PROGRAM MAIN_LINE2
VAR
	traError			: BOOL;
	traInitDone			: BOOL;
	bModeOff			: BOOL;
	bModeManual			: BOOL := TRUE;
	bModeAuto			: BOOL;
	Err_T				: R_TRIG;
	Wrn_T				: R_TRIG;
	fbtimer				: TON;
	fbTimerSirens		: TON;
	Run_T				: R_TRIG;
	Stop_T				: R_TRIG;
	k,k1				: INT;
	nState				: INT;
	nState1				: INT;
	nStateEmr			: INT;
	bFaultFlag			: BOOL;
	nstateStop			: INT;
	fbTimerStop			: TON;
	timerStop			: ton;
	timerReset			: TON;
	thne				: INT;
	nState2				: INT;
	Reset_T				: R_TRIG;
	fbEventlogger		: FB_Eventlogger;
	bWriteAlarm			: BOOL;
END_VAR

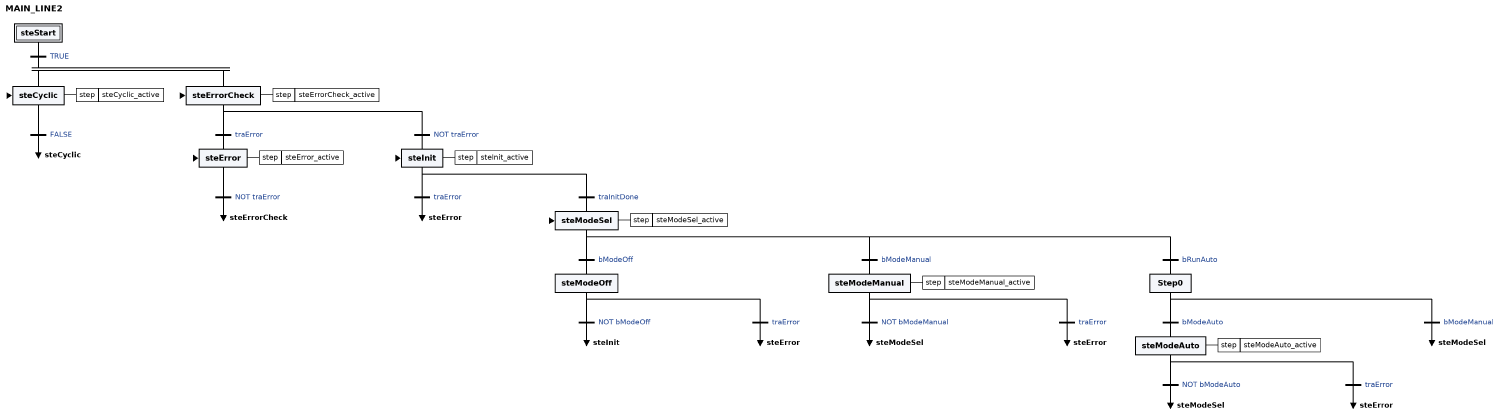
INITIAL_STEP steStart:
END_STEP
TRANSITION FROM steStart TO (steCyclic, steErrorCheck)
    := TRUE;
END_TRANSITION
STEP steCyclic:
    steCyclic_active(N);  // step action
END_STEP
TRANSITION FROM steCyclic TO steCyclic
    := FALSE;
END_TRANSITION
STEP steErrorCheck:
    steErrorCheck_active(N);  // step action
END_STEP
TRANSITION FROM steErrorCheck TO steError
    := traError;
END_TRANSITION
STEP steError:
    steError_active(N);  // step action
END_STEP
TRANSITION FROM steError TO steErrorCheck
    := NOT traError;
END_TRANSITION
TRANSITION FROM steErrorCheck TO steInit
    := NOT traError;
END_TRANSITION
STEP steInit:
    steInit_active(N);  // step action
END_STEP
TRANSITION FROM steInit TO steError
    := traError;
END_TRANSITION
TRANSITION FROM steInit TO steModeSel
    := traInitDone;
END_TRANSITION
STEP steModeSel:
    steModeSel_active(N);  // step action
END_STEP
TRANSITION FROM steModeSel TO steModeOff
    := bModeOff;
END_TRANSITION
STEP steModeOff:
END_STEP
TRANSITION FROM steModeOff TO steInit
    := NOT bModeOff;
END_TRANSITION
TRANSITION FROM steModeOff TO steError
    := traError;
END_TRANSITION
TRANSITION FROM steModeSel TO steModeManual
    := bModeManual;
END_TRANSITION
STEP steModeManual:
    steModeManual_active(N);  // step action
END_STEP
TRANSITION FROM steModeManual TO steModeSel
    := NOT bModeManual;
END_TRANSITION
TRANSITION FROM steModeManual TO steError
    := traError;
END_TRANSITION
TRANSITION FROM steModeSel TO Step0
    := bRunAuto;
END_TRANSITION
STEP Step0:
END_STEP
TRANSITION FROM Step0 TO steModeAuto
    := bModeAuto;
END_TRANSITION
TRANSITION FROM Step0 TO steModeSel
    := bModeManual;
END_TRANSITION
STEP steModeAuto:
    steModeAuto_active(N);  // step action
END_STEP
TRANSITION FROM steModeAuto TO steModeSel
    := NOT bModeAuto;
END_TRANSITION
TRANSITION FROM steModeAuto TO steError
    := traError;
END_TRANSITION

ACTION ListError:
Err_T(CLK := bError2);
Wrn_T(CLK := bWarning2);
GetLocalSystemTime(bEnable := 1,);
IF a2 > 100 THEN
	a2 := 100;
END_IF
		
CASE nState OF 
	0:
		IF Err_T.Q THEN
			nState := 1;
		ELSIF Wrn_T.Q THEN
			bWrn2 := true;
			nState := 10;
		END_IF
	1:
		CASE nErrorID OF	
			23:
				stErrorTxt2 := "E1_2.Lỗi hết hũ trạm 2 [kiểm tra U1I2-4]";
				stErrorTxt3 := 'E1_2.The jar is empty line 2 [check U1I2-4]';
				fbEventlogger(eventClass := TC_EVENTS.Entobel.Event23.uuidEventClass, nEventID := DINT_TO_UDINT(nErrorID));
			24:
				stErrorTxt2 := "E2_2.Lỗi hũ bị kẹt trạm 2 [kiểm tra U1I2-8]";
				stErrorTxt3 := 'E2_2.The jar  is trapped line 2 [check U1I2-8]';
				fbEventlogger(eventClass := TC_EVENTS.Entobel.Event24.uuidEventClass, nEventID := DINT_TO_UDINT(nErrorID));
			25:
				stErrorTxt2 := "E3_2.Lỗi ben chặn hũ trên rút về trạm 2 [kiểm tra U1I2-5]" ;
				stErrorTxt3 := 'E3_2.The upper cylinder retract  is faulty line 2 [check U1I2-5]';
				fbEventlogger(eventClass := TC_EVENTS.Entobel.Event25.uuidEventClass, nEventID := DINT_TO_UDINT(nErrorID));
			26:
				stErrorTxt2 := "E4_2.Lỗi ben chặn hũ dưới rút về trạm 2 [kiểm tra U1I2-6]";
				stErrorTxt3 := 'E4_2.The lower cylinder retract  is faulty line 2 [check U1I2-6]';
				fbEventlogger(eventClass := TC_EVENTS.Entobel.Event26.uuidEventClass, nEventID := DINT_TO_UDINT(nErrorID));
			27:
				stErrorTxt2 := "E5_2.Lỗi ben chặn hũ dưới đẩy ra trạm 2 [kiểm tra U1I2-7]";
				stErrorTxt3 := 'E5_2.The lower cylinder extend  is faulty line 2 [check U1I2-7]';
				fbEventlogger(eventClass := TC_EVENTS.Entobel.Event27.uuidEventClass, nEventID := DINT_TO_UDINT(nErrorID));
			28:
				stErrorTxt2 := "E6_2.Lỗi biến tần đảo thức ăn trạm 2 [kiểm tra biến tần 1]";
				stErrorTxt3 := 'E6_2.The inverter of agitator motor fault line 2 [check inverter 1]';
				fbEventlogger(eventClass := TC_EVENTS.Entobel.Event28.uuidEventClass, nEventID := DINT_TO_UDINT(nErrorID));
			29:
				stErrorTxt2 := "E7_2.Lỗi driver chia thức ăn trạm 2 [kiểm tra driver 1]";
				stErrorTxt3 := 'E7_2.The driver of dispenser motor fault line 2 [check driver 1]';
				fbEventlogger(eventClass := TC_EVENTS.Entobel.Event29.uuidEventClass, nEventID := DINT_TO_UDINT(nErrorID));
			30:
				stErrorTxt2 := "E8_2.Lỗi ben chặn sâu rút về trạm 2 [kiểm tra U1I3-1]";
				stErrorTxt3 := 'E8_2.The cylinder blocking worm retract is faulty line 2 [check U1I3-1]';
				fbEventlogger(eventClass := TC_EVENTS.Entobel.Event30.uuidEventClass, nEventID := DINT_TO_UDINT(nErrorID));
			31:
				stErrorTxt2 := "E9_2.Lỗi biến tần phểu rung sâu trạm 2 [kiểm tra biến tần 2]";
				stErrorTxt3 := 'E9_2.The inverter of vibrating funnel fault line 2 [check inverter 2]';
				fbEventlogger(eventClass := TC_EVENTS.Entobel.Event31.uuidEventClass, nEventID := DINT_TO_UDINT(nErrorID));
			32:
				stErrorTxt2 := "E10_2.Lỗi hết nắp trạm 2 [kiểm tra U1I3-2]";
				stErrorTxt3 := 'E10_2.The lid is empty line 2 [check U1I3-2]';
				fbEventlogger(eventClass := TC_EVENTS.Entobel.Event32.uuidEventClass, nEventID := DINT_TO_UDINT(nErrorID));
			33:
				stErrorTxt2 := "E11_2.Lỗi ben chặn nắp rút về trạm 2 [kiểm tra U1I3-3]";
				stErrorTxt3 := 'E11_2.The cylinder blocking the lid retract is faulty line 2 [check U1I3-3]';
				fbEventlogger(eventClass := TC_EVENTS.Entobel.Event33.uuidEventClass, nEventID := DINT_TO_UDINT(nErrorID));
			34:
				stErrorTxt2 := "E12_2.Lỗi ben chặn nắp đẩy ra trạm 2 [kiểm tra U1I3-4]";
				stErrorTxt3 := 'E12_2.The cylinder blocking the lid extend is faulty line 2 [check U1I3-4]';
				fbEventlogger(eventClass := TC_EVENTS.Entobel.Event34.uuidEventClass, nEventID := DINT_TO_UDINT(nErrorID));
			35:
				stErrorTxt2 := "E13_2.Lỗi ben hút/thả nắp rút ra trạm 2 [kiểm tra U1I3-5]";
				stErrorTxt3 := 'E13_2.The cylinder sucking the lid retract is faulty line 2 [check U1I3-5]';
				fbEventlogger(eventClass := TC_EVENTS.Entobel.Event35.uuidEventClass, nEventID := DINT_TO_UDINT(nErrorID));
			36:
				stErrorTxt2 := "E14_2.Lỗi ben hút/thả nắp đẩy ra trạm 2 [kiểm tra U1I3-6]";
				stErrorTxt3 := 'E14_2.The cylinder sucking the lid extend is faulty line 2 [check U1I3-6]';
				fbEventlogger(eventClass := TC_EVENTS.Entobel.Event36.uuidEventClass, nEventID := DINT_TO_UDINT(nErrorID));
			37:
				stErrorTxt2 := "E15_2.Lỗi ben dập nắp rút về trạm 2 [kiểm tra U1I3-8]";
				stErrorTxt3 := 'E15_2.The cylinder pressing the lid retract is faulty line 2 [check U1I3-8]';
				fbEventlogger(eventClass := TC_EVENTS.Entobel.Event37.uuidEventClass, nEventID := DINT_TO_UDINT(nErrorID));
			38:
				stErrorTxt2 := "E16_2.Lỗi ben dập nắp đẩy ra trạm 2 [kiểm tra U1I4-1]";
				stErrorTxt3 := 'E16_2.The cylinder pressing the lid extend is faulty line 2 [check U1I4-1]';
				fbEventlogger(eventClass := TC_EVENTS.Entobel.Event38.uuidEventClass, nEventID := DINT_TO_UDINT(nErrorID));
			39:
				stErrorTxt2 := "E17_2.Lỗi ben lượt ra/vào Rút về trạm 2 [kiểm tra U1I4-2]";
				stErrorTxt3 := 'E17_2.The comb cylinder retract is faulty line 2 [check U1I4-2]';
				fbEventlogger(eventClass := TC_EVENTS.Entobel.Event39.uuidEventClass, nEventID := DINT_TO_UDINT(nErrorID));
			40:
				stErrorTxt2 := "E18_2.Lỗi ben lượt ra/vào đẩy ra trạm 2 [kiểm tra U1I4-3]";
				stErrorTxt3 := 'E18_2.The comb cylinder extend is faulty line 2 [check U1I4-3]';
				fbEventlogger(eventClass := TC_EVENTS.Entobel.Event40.uuidEventClass, nEventID := DINT_TO_UDINT(nErrorID));
			41:
				stErrorTxt2 := "E19_2.Lỗi ben kẹp hũ rút về trạm 2 [kiểm tra U1I4-6]";
				stErrorTxt3 := 'E19_2.The clap cylinder retract is faulty line 2 [check U1I4-6]';
				fbEventlogger(eventClass := TC_EVENTS.Entobel.Event41.uuidEventClass, nEventID := DINT_TO_UDINT(nErrorID));
			42:
				stErrorTxt2 := "E20_2.Lỗi ben kẹp hũ đẩy ra trạm 2 [kiểm tra U1I4-7]";	
				stErrorTxt3 := 'E20_2.The clap cylinder extend is faulty 2 [check U1I4-4]';
				fbEventlogger(eventClass := TC_EVENTS.Entobel.Event42.uuidEventClass, nEventID := DINT_TO_UDINT(nErrorID));
			43:
				stErrorTxt2 := "E21_2.Lỗi ben di chuyển lượt rút về trạm 2 [kiểm tra U1I4-4]";	
				stErrorTxt3 := 'E21_2.The cylinder moving comb retract is faulty line 2 [check U1I4-4]';
				fbEventlogger(eventClass := TC_EVENTS.Entobel.Event43.uuidEventClass, nEventID := DINT_TO_UDINT(nErrorID));
			44:
				stErrorTxt2 := "E22_2.Lỗi ben di chuyển lượt đẩy ra trạm 2 [kiểm tra U1I4-5]";	
				stErrorTxt3 := 'E22_2.The cylinder moving comb extend is faulty line 2 [check U1I4-5]';
				fbEventlogger(eventClass := TC_EVENTS.Entobel.Event44.uuidEventClass, nEventID := DINT_TO_UDINT(nErrorID));
			46:
				stErrorTxt2 := "E23_2.Lỗi mất hũ khi đang cân thức ăn trạm 2 [kiểm tra U1I4-8]";
				stErrorTxt3 := 'E23_2.The jar is missed when weighting food line 2 [check U1I4-8]';
				fbEventlogger(eventClass := TC_EVENTS.Entobel.Event46.uuidEventClass, nEventID := DINT_TO_UDINT(nErrorID));
			48:
				stErrorTxt2 := "E24_2.Lỗi mất hũ khi đang cân sâu trạm 2 [kiểm tra U1I5-1]";
				stErrorTxt3 := 'E24_2.The jar is missed when weighting larvae line 2 [check U1I5-1]';
				fbEventlogger(eventClass := TC_EVENTS.Entobel.Event48.uuidEventClass, nEventID := DINT_TO_UDINT(nErrorID));
			50:
				stErrorTxt2 := "E25_2.Lỗi hút không được nắp trạm 2 [kiểm tra U1I3-7]";
				stErrorTxt3 := 'E25_2.Failed to suction the lid  line 2 [check U1I3-7]';
				fbEventlogger(eventClass := TC_EVENTS.Entobel.Event50.uuidEventClass, nEventID := DINT_TO_UDINT(nErrorID));
			52:
				stErrorTxt2 := "E26_2.Lỗi nắp đã được hút 2 [kiểm tra U1I3-7]";	
				stErrorTxt3 := 'E26_2.The lid is still on the valve line 2 [check U1I3-7]';
				fbEventlogger(eventClass := TC_EVENTS.Entobel.Event52.uuidEventClass, nEventID := DINT_TO_UDINT(nErrorID));
			53:
				stErrorTxt2 := "E27_2.Lỗi an toàn cửa 1 [kiểm tra U1I7-8]";	
				stErrorTxt3 := 'E27_2.The safety door 1 is error [check U1I7-8]';
			54:
				stErrorTxt2 := "E28_2.Lỗi an toàn cửa 2 [kiểm tra U1I7-9]";
				stErrorTxt3 := 'E28_2.The safety door 2 is error [check U1I7-9]';
			55:
				stErrorTxt2 := "E29_2.Lỗi an toàn cửa 3 [kiểm tra U1I7-10]";
				stErrorTxt3 := 'E29_2.The safety door 3 is error [check U1I7-10]';
			58: 
				stErrorTxt2 := "E30_2.Lỗi quá cân thức ăn trạm 2 [kiểm tra cân thức ăn]";
				stErrorTxt3 := 'E30_2.Overload weightfood line 2 [check weightfood]';
				fbEventlogger(eventClass := TC_EVENTS.Entobel.Event58.uuidEventClass, nEventID := DINT_TO_UDINT(nErrorID));
			59: 
				stErrorTxt2 := "E31_2.Lỗi quá cân sâu trạm 2 [kiểm tra cân sâu]";
				stErrorTxt3 := 'E31_2.Overload weightlarvae line 2 [check weightlarvae]';
				fbEventlogger(eventClass := TC_EVENTS.Entobel.Event59.uuidEventClass, nEventID := DINT_TO_UDINT(nErrorID));
			61:
				stErrorTxt2 := "E32_2.Lỗi ben hút/thả hũ đẩy ra trạm 2 [kiểm tra U1I7-12]";
				stErrorTxt3 := 'E32_2.The cylinder sucking the jar is faulty line 2 [check U1I7-12]';
				fbEventlogger(eventClass := TC_EVENTS.Entobel.Event61.uuidEventClass, nEventID := DINT_TO_UDINT(nErrorID));
			62:
				stErrorTxt2 := "E33_2.Lỗi Modbus thiết bị 1";
				stErrorTxt3 := 'E33_2.Error Modbus device 1';
				fbEventlogger(eventClass := TC_EVENTS.Entobel.Event62.uuidEventClass, nEventID := DINT_TO_UDINT(nErrorID));
			63:
				stErrorTxt2 := "E34_2.Lỗi Modbus thiết bị 2";
				stErrorTxt3 := 'E34_2.Error Modbus device 2';
				fbEventlogger(eventClass := TC_EVENTS.Entobel.Event63.uuidEventClass, nEventID := DINT_TO_UDINT(nErrorID));
			64:
				stErrorTxt2 := "E35_2.Lỗi Modbus thiết bị 3";
				stErrorTxt3 := 'E35_2.Error Modbus device 3';
			67:
				stErrorTxt2 := "E36_2.Lỗi Modbus thiết bị 6";
				stErrorTxt3 := 'E36_2.Error Modbus device 6';
				fbEventlogger(eventClass := TC_EVENTS.Entobel.Event67.uuidEventClass, nEventID := DINT_TO_UDINT(nErrorID));
			71:
				stErrorTxt2 := "E37_2.Lỗi đầu cân thức ăn Laumas";
				stErrorTxt3 := 'E37_2.Error Laumas 1';
				fbEventlogger(eventClass := TC_EVENTS.Entobel.Event71.uuidEventClass, nEventID := DINT_TO_UDINT(nErrorID));
			72:
				stErrorTxt2 := "E38_2.Lỗi đầu cân sâu Laumas";
				stErrorTxt3 := 'E38_2.Error Laumas 2';
				fbEventlogger(eventClass := TC_EVENTS.Entobel.Event72.uuidEventClass, nEventID := DINT_TO_UDINT(nErrorID));
			74:
				stErrorTxt2 := "E39_2.Lỗi ben chặn sâu đẩy ra trạm 2 [kiểm tra U1I3-1]";
				stErrorTxt3 := 'E39_2.The cylinder blocking worm extend  is faulty line 2';
				fbEventlogger(eventClass := TC_EVENTS.Entobel.Event74.uuidEventClass, nEventID := DINT_TO_UDINT(nErrorID));
			75:
				stErrorTxt2 := "E40_2.Lỗi thiếu khí đầu vào [kiểm tra U1I7-13]";
				stErrorTxt3 := 'E40_2.Error of lack of input air [check U1I7-13]';	
			78:
				stErrorTxt2 := "E41_2.Lỗi hết thức ăn trạm 2";
				stErrorTxt3 := 'E41_2.Error running out of food line 2';
				fbEventlogger(eventClass := TC_EVENTS.Entobel.Event77.uuidEventClass, nEventID := DINT_TO_UDINT(nErrorID));	
			79:
				stErrorTxt2 := "E42_2.Lỗi hết sâu trạm 2";
				stErrorTxt3 := 'E42_2.Error running out of larvae line 2';
				fbEventlogger(eventClass := TC_EVENTS.Entobel.Event79.uuidEventClass, nEventID := DINT_TO_UDINT(nErrorID));	
			98:
				stErrorTxt2 := "E98_2.Dừng khẩn [kiểm tra Emergency]"; 
				stErrorTxt3 := 'E98_2.Emergency Stop [check Emergency]';
			99: 
				stErrorTxt2 := "E99_2.Lỗi biến tần băng tải đầu ra [kiểm tra biến tần 3]";
				stErrorTxt3 := 'E99_2.The inverter of conveyor ouy [check inverter 3]';
		END_CASE
		IF a2 <> 1 THEN
			FOR	k := a2 TO 2 BY -1 DO
				nErrorIDList2[k].nErrorID 	 := nErrorIDList2[k-1].nErrorID;
				nErrorIDList2[k].ErrorTime   := nErrorIDList2[k-1].ErrorTime;
				nErrorIDList2[k].ErrorStatus := nErrorIDList2[k-1].ErrorStatus;	
			END_FOR		
		END_IF 
		nErrorIDList2[1].nErrorID := nErrorID;
		nErrorIDList2[1].ErrorTime := SYSTEMTIME_TO_DT(GetLocalSystemTime.systemTime);
		nErrorIDList2[1].ErrorStatus := 1;
		nStatus2	:= 'ERROR';
		a2 := a2 + 1;
		bWarning := FALSE;
		nState := 2;
	2:
		bWriteAlarm	:= TRUE;
		IF nErrorID = 53 THEN
			bTo_alarm_side2 := FALSE;
		ELSIF nErrorID = 54 THEN
			bTo_alarm_side2 := FALSE;
		ELSIF nErrorID = 55 THEN
			bTo_alarm_side2 := FALSE;
		ELSIF nErrorID = 64 THEN
			bTo_alarm_side2 := FALSE;
		ELSIF nErrorID = 75 THEN
			bTo_alarm_side2 := FALSE;
		ELSIF nErrorID = 98 THEN
			bTo_alarm_side2 := FALSE;
		ELSIF nErrorID = 99 THEN
			bTo_alarm_side2 := FALSE;
		ELSE 	
			bTo_alarm_side2 := TRUE;
		END_IF
		bSirens := TRUE;
		nState := 3;
	3:
		IF NOT bError2 THEN
			nState 	:= 0;
		END_IF
	10:
		CASE nWarningID OF
			108:
				stWarningTxt2 := "W1_2.Cảnh báo hết hũ trạm 2 [kiểm tra U1I2-4]";
				stWarningTxt3 := 'W1_2.Warning out of jar line 2 [check U1I2-4]';
				fbEventlogger(eventClass := TC_EVENTS.Entobel.Event108.uuidEventClass, nEventID := DINT_TO_UDINT(nWarningID));
			109:
				stWarningTxt2 := "W2_2.Cảnh báo hết nắp trạm 2 [kiểm tra U1I3-2]";
				stWarningTxt3 := 'W2_2.Warning out of lid line 2 [check U1I3-2]';
				fbEventlogger(eventClass := TC_EVENTS.Entobel.Event109.uuidEventClass, nEventID := DINT_TO_UDINT(nWarningID));
			110:
				stWarningTxt2 := "W3_2.Cảnh báo hết thức ăn trạm 2";
				stWarningTxt3 := 'W3_2.Warning running out of food line 2';
				fbEventlogger(eventClass := TC_EVENTS.Entobel.Event110.uuidEventClass, nEventID := DINT_TO_UDINT(nWarningID));
			111:
				stWarningTxt2 := "W4_2.Cảnh báo cân quá khối lượng thức ăn trạm 2";
				stWarningTxt3 := 'W4_2.Warning food weight exceeds limit line 2';
				fbEventlogger(eventClass := TC_EVENTS.Entobel.Event111.uuidEventClass, nEventID := DINT_TO_UDINT(nWarningID));
			112:
				stWarningTxt2 := "W5_2.Cảnh báo hết sâu trạm 2";
				stWarningTxt3 := 'W5_2.Warning running out of larvae line 2';
				fbEventlogger(eventClass := TC_EVENTS.Entobel.Event112.uuidEventClass, nEventID := DINT_TO_UDINT(nWarningID));
			113:
				stWarningTxt2 := "W6_2.Canh bao can qua khoi luong sau tram 2";
				stWarningTxt3 := 'W6_2.Warning larvae weight exceeds limit line 2';
				fbEventlogger(eventClass := TC_EVENTS.Entobel.Event113.uuidEventClass, nEventID := DINT_TO_UDINT(nWarningID));
			114:
				stWarningTxt2 := "W7_2.Cảnh báo dập nắp không vô trạm 2 [kiểm tra U1I4-1]";
				stWarningTxt3 := 'W7_2.Warning do not press lid inward line 2 [check U1I4-1]';
				fbEventlogger(eventClass := TC_EVENTS.Entobel.Event114.uuidEventClass, nEventID := DINT_TO_UDINT(nWarningID));
			115:
				stWarningTxt2 := "W8_2.Cảnh báo mất kết nối với PC Advantech [kiểm tra PC]";
				stWarningTxt3 := 'W8_2.Warning disconnect to PC Advantech [check PC]';	
		END_CASE
		IF a2 <> 1 THEN
			FOR	k := a2 TO 2 BY -1 DO
				nErrorIDList2[k].nErrorID 	 := nErrorIDList2[k-1].nErrorID;
				nErrorIDList2[k].ErrorTime   := nErrorIDList2[k-1].ErrorTime;
				nErrorIDList2[k].ErrorStatus := nErrorIDList2[k-1].ErrorStatus;			
			END_FOR		
		END_IF 
		nErrorIDList2[1].nErrorID := nWarningID;
		nErrorIDList2[1].ErrorTime := SYSTEMTIME_TO_DT(GetLocalSystemTime.systemTime);
		nErrorIDList2[1].ErrorStatus := 1;
		nStatus1	:= 'WARNING';
		a2 := a2 + 1;
		nState := 11;
	11:
		bWriteAlarm	:= TRUE;
		bSirens := TRUE;
		nState := 12;
	12:
		bWarning2 := FALSE;
		nState := 0;		
END_CASE

IF bclearall THEN
	FOR k := 1 TO 100 DO
		AlarmList2[1,k] := "";
		AlarmList2[2,k] := "";	
		AlarmList2[3,k] := "";
		AlarmList2[4,k] := "";	
		AlarmList4[1,k] := '';
		AlarmList4[2,k] := '';	
		AlarmList4[3,k] := '';
		AlarmList4[4,k] := '';	
	END_FOR
	a2 := 1;
END_IF
END_ACTION

ACTION Reset_active:
PR_Line02.Reset();
END_ACTION

ACTION steCyclic_active:
PR_Line02();
ListError();;
GetLocalSystemTime(bEnable := 1,);
SystemTimeFull 	:= SYSTEMTIME_TO_STRING(in := GetLocalSystemTime.systemTime);
PRG_MainRecipe1_1();

IF bError2 THEN
	traError := true;
END_IF

IF NOT bEmer THEN
	traError := TRUE;
END_IF
IF bWriteAlarm	THEN
FOR k1 := 1 TO 100 DO
	AlarmList2[1,k1] 	:= INT_TO_WSTRING(nErrorIDList2[k1].nErrorID);
	AlarmList4[1,k1]	:= INT_TO_STRING(nErrorIDList2[k1].nErrorID);
	AlarmList2[4,k1] 	:= STRING_TO_WSTRING(MID(STR := DT_TO_STRING(nErrorIDList2[k1].ErrorTime),LEN := 19, POS := 4));
	AlarmList4[4,k1] 	:= MID(STR := DT_TO_STRING(nErrorIDList2[k1].ErrorTime),LEN := 19, POS := 4);
	IF nErrorIDList2[k1].ErrorStatus = 1 THEN
		AlarmList2[3,k1] := "Active";
		AlarmList4[3,k1] := 'Active';
	ELSE
		AlarmList2[3,k1] := "Release";
		AlarmList4[3,k1] := 'Release';
	END_IF
	CASE nErrorIDList2[k1].nErrorID OF 
			0:
				AlarmList2[4,k1] 	:= "";
				AlarmList2[3,k1] 	:= "";
				AlarmList4[4,k1] 	:= '';
				AlarmList4[3,k1] 	:= '';
			23:
				AlarmList2[2,k1] := "E1_2.Lỗi hết hũ trạm 2 [kiểm tra U1I2-4]";
				AlarmList4[2,k1] := 'E1_2.The jar is empty line 2 [check U1I2-4]';
			24:
				AlarmList2[2,k1] := "E2_2.Lỗi hũ bị kẹt trạm 2 [kiểm tra U1I2-8]";
				AlarmList4[2,k1] := 'E2_2.The jar  is trapped line 2 [check U1I2-8]';
			25:
				AlarmList2[2,k1] := "E3_2.Lỗi ben chặn hũ trên rút về trạm 2 [kiểm tra U1I2-5]" ;
				AlarmList4[2,k1] := 'E3_2.The upper cylinder retract  is faulty line 2 [check U1I2-5]';
			26:
				AlarmList2[2,k1] := "E4_2.Lỗi ben chặn hũ dưới rút về trạm 2 [kiểm tra U1I2-6]";
				AlarmList4[2,k1] := 'E4_2.The lower cylinder retract  is faulty line 2 [check U1I2-6]';
			27:
				AlarmList2[2,k1] := "E5_2.Lỗi ben chặn hũ dưới đẩy ra trạm 2 [kiểm tra U1I2-7]";
				AlarmList4[2,k1] := 'E5_2.The lower cylinder extend  is faulty line 2 [check U1I2-7]';
			28:
				AlarmList2[2,k1] := "E6_2.Lỗi biến tần đảo thức ăn trạm 2 [kiểm tra biến tần 1]";
				AlarmList4[2,k1] := 'E6_2.The inverter of agitator motor fault line 2 [check inverter 1]';
			29:
				AlarmList2[2,k1] := "E7_2.Lỗi driver chia thức ăn trạm 2 [kiểm tra driver 1]";
				AlarmList4[2,k1] := 'E7_2.The driver of dispenser motor fault line 2 [check driver 1]';
			30:
				AlarmList2[2,k1] := "E8_2.Lỗi ben chặn sâu rút về trạm 2 [kiểm tra U1I3-1]";
				AlarmList4[2,k1] := 'E8_2.The cylinder blocking worm retract is faulty line 2 [check U1I3-1]';
			31:
				AlarmList2[2,k1] := "E9_2.Lỗi biến tần phểu rung sâu trạm 2 [kiểm tra biến tần 2]";
				AlarmList4[2,k1] := 'E9_2.The inverter of vibrating funnel fault line 2 [check inverter 2]';
			32:
				AlarmList2[2,k1] := "E10_2.Lỗi hết nắp trạm 2 [kiểm tra U1I3-2]";
				AlarmList4[2,k1] := 'E10_2.The lid is empty line 2 [check U1I3-2]';
			33:
				AlarmList2[2,k1] := "E11_2.Lỗi ben chặn nắp rút về trạm 2 [kiểm tra U1I3-3]";
				AlarmList4[2,k1] := 'E11_2.The cylinder blocking the lid retract is faulty line 2 [check U1I3-3]';
			34:
				AlarmList2[2,k1] := "E12_2.Lỗi ben chặn nắp đẩy ra trạm 2 [kiểm tra U1I3-4]";
				AlarmList4[2,k1] := 'E12_2.The cylinder blocking the lid extend is faulty line 2 [check U1I3-4]';
			35:
				AlarmList2[2,k1] := "E13_2.Lỗi ben hút/thả nắp rút ra trạm 2 [kiểm tra U1I3-5]";
				AlarmList4[2,k1] := 'E13_2.The cylinder sucking the lid retract is faulty line 2 [check U1I3-5]';
			36:
				AlarmList2[2,k1] := "E14_2.Lỗi ben hút/thả nắp đẩy ra trạm 2 [kiểm tra U1I3-6]";
				AlarmList4[2,k1] := 'E14_2.The cylinder sucking the lid extend is faulty line 2 [check U1I3-6]';
			37:
				AlarmList2[2,k1] := "E15_2.Lỗi ben dập nắp rút về trạm 2 [kiểm tra U1I3-8]";
				AlarmList4[2,k1] := 'E15_2.The cylinder pressing the lid retract is faulty line 2 [check U1I3-8]';
			38:
				AlarmList2[2,k1] := "E16_2.Lỗi ben dập nắp đẩy ra trạm 2 [kiểm tra U1I4-1]";
				AlarmList4[2,k1] := 'E16_2.The cylinder pressing the lid extend is faulty line 2 [check U1I4-1]';
			39:
				AlarmList2[2,k1] := "E17_2.Lỗi ben lượt ra/vào Rút về trạm 2 [kiểm tra U1I4-2]";
				AlarmList4[2,k1] := 'E17_2.The comb cylinder retract is faulty line 2 [check U1I4-2]';
			40:
				AlarmList2[2,k1] := "E18_2.Lỗi ben lượt ra/vào đẩy ra trạm 2 [kiểm tra U1I4-3]";
				AlarmList4[2,k1] := 'E18_2.The comb cylinder extend is faulty line 2 [check U1I4-3]';
			41:
				AlarmList2[2,k1] := "E19_2.Lỗi ben kẹp hũ rút về trạm 2 [kiểm tra U1I4-6]";
				AlarmList4[2,k1] := 'E19_2.The clap cylinder retract is faulty line 2 [check U1I4-6]';
			42:
				AlarmList2[2,k1] := "E20_2.Lỗi ben kẹp hũ đẩy ra trạm 2 [kiểm tra U1I4-7]";	
				AlarmList4[2,k1] := 'E20_2.The clap cylinder extend is faulty 2 [check U1I4-4]';
			43:
				AlarmList2[2,k1] := "E21_2.Lỗi ben di chuyển lượt rút về trạm 2 [kiểm tra U1I4-4]";	
				AlarmList4[2,k1] := 'E21_2.The cylinder moving comb retract is faulty line 2 [check U1I4-4]';
			44:
				AlarmList2[2,k1] := "E22_2.Lỗi ben di chuyển lượt đẩy ra trạm 2 [kiểm tra U1I4-5]";	
				AlarmList4[2,k1] := 'E22_2.The cylinder moving comb extend is faulty line 2 [check U1I4-5]';
			46:
				AlarmList2[2,k1] := "E23_2.Lỗi mất hũ khi đang cân thức ăn trạm 2 [kiểm tra U1I4-8]";
				AlarmList4[2,k1] := 'E23_2.The jar is missed when weighting food line 2 [check U1I4-8]';
			48:
				AlarmList2[2,k1] := "E24_2.Lỗi mất hũ khi đang cân sâu trạm 2 [kiểm tra U1I5-1]";
				AlarmList4[2,k1] := 'E24_2.The jar is missed when weighting larvae line 2 [check U1I5-1]';
			50:
				AlarmList2[2,k1] := "E25_2.Lỗi hút không được nắp trạm 2 [kiểm tra U1I3-7]";
				AlarmList4[2,k1] := 'E25_2.Failed to suction the lid  line 2 [check U1I3-7]';
			52:
				AlarmList2[2,k1] := "E26_2.Lỗi nắp đã được hút 2 [kiểm tra U1I3-7]";	
				AlarmList4[2,k1] := 'E26_2.The lid is still on the valve line 2 [check U1I3-7]';
			53:
				AlarmList2[2,k1] := "E27_2.Lỗi an toàn cửa 1 [kiểm tra U1I7-8]";	
				AlarmList4[2,k1] := 'E27_2.The safety door 1 is error [check U1I7-8]';
			54:
				AlarmList2[2,k1] := "E28_2.Lỗi an toàn cửa 2 [kiểm tra U1I7-9]";
				AlarmList4[2,k1] := 'E28_2.The safety door 2 is error [check U1I7-9]';
			55:
				AlarmList2[2,k1] := "E29_2.Lỗi an toàn cửa 3 [kiểm tra U1I7-10]";
				AlarmList4[2,k1] := 'E29_2.The safety door 3 is error [check U1I7-10]';
			58: 
				AlarmList2[2,k1] := "E30_2.Lỗi quá cân thức ăn trạm 2 [kiểm tra cân thức ăn]";
				AlarmList4[2,k1] := 'E30_2.Overload weightfood line 2 [check weightfood]';
			59: 
				AlarmList2[2,k1] := "E31_2.Lỗi quá cân sâu trạm 2 [kiểm tra cân sâu]";
				AlarmList4[2,k1] := 'E31_2.Overload weightlarvae line 2 [check weightlarvae]';
			61:
				AlarmList2[2,k1] := "E32_2.Lỗi ben hút/thả hũ đẩy ra trạm 2 [kiểm tra U1I7-12]";
				AlarmList4[2,k1] := 'E32_2.The cylinder sucking the jar is faulty line 2 [check U1I7-12]';
			62:
				AlarmList2[2,k1] := "E33_2.Lỗi Modbus thiết bị 1";
				AlarmList4[2,k1] := 'E33_2.Error Modbus device 1';
			63:
				AlarmList2[2,k1] := "E34_2.Lỗi Modbus thiết bị 2";
				AlarmList4[2,k1] := 'E34_2.Error Modbus device 2';
			64:
				AlarmList2[2,k1] := "E35_2.Lỗi Modbus thiết bị 3";
				AlarmList4[2,k1] := 'E35_2.Error Modbus device 3';
			67:
				AlarmList2[2,k1] := "E36_2.Lỗi Modbus thiết bị 6";
				AlarmList4[2,k1] := 'E36_2.Error Modbus device 6';
			71:
				AlarmList2[2,k1] := "E37_2.Lỗi đầu cân thức ăn Laumas";
				AlarmList4[2,k1] := 'E37_2.Error Laumas 1';
			72:
				AlarmList2[2,k1] := "E38_2.Lỗi đầu cân sâu Laumas";
				stErrorTxt3 := 'E38_2.Error Laumas 2';
			74:
				AlarmList2[2,k1] := "E39_2.Lỗi ben chặn sâu đẩy ra trạm 2 [kiểm tra U1I3-1]";
				AlarmList4[2,k1] := 'E39_2.The cylinder blocking worm extend  is faulty line 2';
			75:
				AlarmList2[2,k1] := "E40_2.Lỗi thiếu khí đầu vào [kiểm tra U1I7-13]";
				AlarmList4[2,k1] := 'E40_2.Error of lack of input air [check U1I7-13]';	
			78:
				AlarmList2[2,k1] := "E41_2.Lỗi hết thức ăn trạm 2";
				AlarmList4[2,k1] := 'E41_2.Error running out of food line 2';	
			79:
				AlarmList2[2,k1] := "E42_2.Lỗi hết sâu trạm 2";
				AlarmList4[2,k1] := 'E42_2.Error running out of larvae line 2';
			98:
				AlarmList2[2,k1] := "E98_2.Dừng khẩn [kiểm tra Emergency]"; 
				AlarmList4[2,k1] := 'E98_2.Emergency Stop [check Emergency]';
			99: 
				AlarmList2[2,k1] := "E99_2.Lỗi biến tần băng tải đầu ra [kiểm tra biến tần 3]";
				AlarmList4[2,k1] := 'E99_2.The inverter of conveyor ouy [check inverter 3]';
			108:
				AlarmList2[2,k1] := "W1_2.Cảnh báo hết hũ trạm 2 [kiểm tra U1I2-4]";
				AlarmList4[2,k1] := 'W1_2.Warning out of jar line 2 [check U1I2-4]';
			109:
				AlarmList2[2,k1] := "W2_2.Cảnh báo hết nắp trạm 2 [kiểm tra U1I3-2]";
				AlarmList4[2,k1] := 'W2_2.Warning out of lid line 2 [check U1I3-2]';
			110:
				AlarmList2[2,k1] := "W3_2.Cảnh báo hết thức ăn trạm 2";
				AlarmList4[2,k1] := 'W3_2.Warning running out of food line 2';
			111:
				AlarmList2[2,k1] := "W4_2.Cảnh báo cân quá khối lượng thức ăn trạm 2";
				AlarmList4[2,k1] := 'W4_2.Warning food weight exceeds limit line 2';
			112:
				AlarmList2[2,k1] := "W5_2.Cảnh báo hết sâu trạm 2";
				AlarmList4[2,k1] := 'W5_2.Warning running out of larvae line 2';
			113:
				AlarmList2[2,k1] := "W6_2.Canh bao can qua khoi luong sau tram 2";
				AlarmList4[2,k1] := 'W6_2.Warning larvae weight exceeds limit line 2';
			114:
				AlarmList2[2,k1] := "W7_2.Cảnh báo dập nắp không vô trạm 2 [kiểm tra U1I4-1]";
				AlarmList4[2,k1] := 'W7_2.Warning do not press lid inward line 2 [check U1I4-1]';
			115:
				AlarmList2[2,k1] := "W8_2.Cảnh báo mất kết nối với PC Advantech [kiểm tra PC]";
				AlarmList4[2,k1] := 'W8_2.Warning disconnect to PC Advantech [check PC]';	
		END_CASE
END_FOR
bWriteAlarm	:= FALSE;
END_IF
END_ACTION

ACTION steError_active:
PR_Line02.Stop();
bStatusStart2 := FALSE;
status := 'ERROR';
bfinish2 := TRUE;
IF a2 > 100 THEN
	a2 := 100;
END_IF
CASE nState2 OF 
	0:
		Reset_T(clk := bReset);
		IF Reset_T.Q THEN
			nState2 := 1;
		END_IF
	1:
		PR_Line02.Reset();
		timerReset(IN := TRUE, PT := T#500MS);
		IF nErrorIDList2[1].ErrorStatus = 1 THEN
			IF i <> 1 THEN
				FOR	k := a2 TO 2 BY -1 DO
				nErrorIDList2[k].nErrorID 	 := nErrorIDList2[k-1].nErrorID;
				nErrorIDList2[k].ErrorTime   := nErrorIDList2[k-1].ErrorTime;
				nErrorIDList2[k].ErrorStatus := nErrorIDList2[k-1].ErrorStatus;		
				END_FOR		
			END_IF 
			nState2 := 2;
		ELSE 
			nState2 := 3;
		END_IF
	2:
		bWriteAlarm	:= TRUE;
		PR_Line02.Reset();
		timerReset(IN := TRUE, PT := T#500MS);
		nErrorIDList2[1].nErrorID := nErrorID;
		nErrorIDList2[1].ErrorTime := SYSTEMTIME_TO_DT(GetLocalSystemTime.systemTime);
		nErrorIDList2[1].ErrorStatus := 0;
		a2 := a2  + 1;	
		nState2 := 3;
	3:
		PR_Line02.Reset();
		timerReset(IN := TRUE, PT := T#500MS);
		IF timerReset.Q THEN
			nState2 := 4;
		END_IF
	4:
		timerReset(IN := FALSE);
		Reset_T(clk := FALSE);
		traError := FALSE;
		nState2 := 0;
END_CASE

IF bReset THEN
	bError2 := FALSE;
	bWarning := FALSE;
	bSirens := FALSE;
	status := 'STOP';
	Error[1] := FALSE;
	Error[2] := FALSE;
	Error[6] := FALSE;
	Error[3] := FALSE;
END_IF

IF NOT bEmer THEN
	PR_Line02.Init();
END_IF

IF bTo_alarm_side2 AND NOT bTo_alarm_side THEN
	VisuElems.CURRENTVISU := 'N_Alarm_1';
	IF VisuElems.CURRENTVISU = 'N_Alarm_1' THEN
		bTo_alarm_side2 := FALSE;
	END_IF
END_IF
END_ACTION

ACTION steErrorCheck_active:

END_ACTION

ACTION steInit_active:
traInitDone := TRUE;
bStatusStart2 := FALSE;
END_ACTION

ACTION steModeAuto_active:
PR_Line02.Auto();
bResetmanual2 := TRUE;
IF bReset THEN
	bWarning2 := FALSE;
	bSirens	  := FALSE;
	bAlarm_Iot := FALSE;
	bWrn2	  := FALSE;
END_IF
END_ACTION

ACTION steModeManual_active:
PR_Line02.Manual();
PR_Line02.Check_reset();
END_ACTION

ACTION steModeSel_active:
IF VisuElems.CURRENTVISU = 'MAIN_LINE2' THEN
	bModeAuto := TRUE;
	bModeManual := FALSE;
END_IF

IF VisuElems.CURRENTVISU = 'N_FoodSupply2' OR VisuElems.CURRENTVISU = 'N_JarSupply2' OR VisuElems.CURRENTVISU = 'N_LidPressing2' OR
	VisuElems.CURRENTVISU = 'N_LidSupply2' OR VisuElems.CURRENTVISU = 'N_Tranfer2' OR VisuElems.CURRENTVISU = 'N_WormWeight2' THEN
	bModeAuto := FALSE;
	bModeManual := TRUE;
END_IF
PR_Line02.check();

IF bStart2 THEN
	bStart2 := FALSE;
END_IF
END_ACTION

END_PROGRAM

(* stored: Version 1.1.0.1, ProductVersion 3.1.4024.12
   POU MAIN_LINE2: Id {13d9e9db-c67d-47e0-8c80-49b58b356c95}, SpecialFunc None
   Action ListError: Id {fa80e241-5590-4bca-b54d-2243a049f4ee}
   Action Reset_active: Id {76f3410b-fd66-4e60-a571-7be8b865ea46}
   Action steCyclic_active: Id {484aa1cc-8f4d-475f-bab8-20cbafd63976}
   Action steError_active: Id {f5815781-baeb-4c8a-9fb1-dffe97744e2c}
   Action steErrorCheck_active: Id {59c5cd30-b7a2-4ec6-ad4f-6ea8d40636d4}
   Action steInit_active: Id {fb88de51-e1ac-4095-a134-d5265480927b}
   Action steModeAuto_active: Id {09639ebb-73bb-48d2-8665-4b9033f2bac8}
   Action steModeManual_active: Id {8b0aac46-9fb9-4437-a4a4-13657bbf58d6}
   Action steModeSel_active: Id {9ef899b0-3f5d-4d53-92eb-527262267d9f} *)
